// TIA Portal V17 export
// export: Created 2024-01-17T02:33:01.6071597Z, ExportSetting None, DisplayName Totally Integrated Automation Portal, DisplayVersion V17 Update 4, DisplayName TIA Portal Openness, DisplayVersion V17 Update 4, DisplayName TIA Portal Version Control Interface, DisplayVersion V17, DisplayName STEP 7 Professional, DisplayVersion V17 Update 4, DisplayName STEP 7 Safety, DisplayVersion V17, DisplayName WinCC Advanced / Unified PC, DisplayVersion V17 Update 4
DATA_BLOCK "FALM"   // DB1016, F_DB
{ S7_Optimized_Access := 'TRUE' }
// stored: AutoNumber false
   VAR
      CQ004XB02 : Bool;
      AN001XJ27 : Bool;
      CQ005XB02 : Bool;
      CQ006XB02 : Bool;
      GH001XB33 : Bool;
      GH001XM01 : Bool;
   END_VAR
BEGIN
END_DATA_BLOCK
